Universal Robots PolyScope program: 05_var_local_01.urp

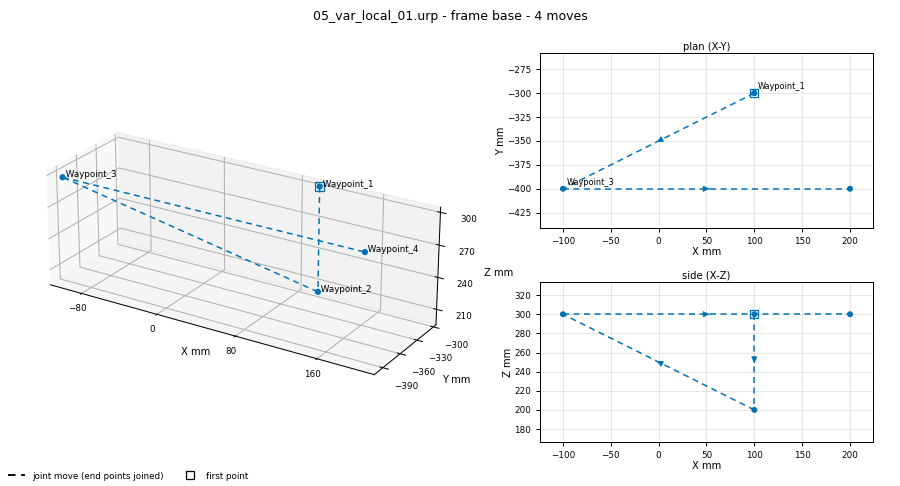
[picture p0: tool path of 05_var_local_01.urp in frame base, 4 of 4 moves have a stored position in this frame; points joined in program order, loops and branches not executed]
Program 05_var_local_01 (installation=default directory=/home/ur/ursim-current/programs/Test_Programs createdIn=5.9.1.1031110 lastSavedIn=5.9.1.1031110 robotSerialNumber=20195599999)
Calibrated DH parameters: a=[0, -0.425, -0.3922, 0, 0, 0]; d=[0.1625, 0, 0, 0.1333, 0.0997, 0.0996]; alpha=[1.570796, 0, 0, 1.570796, -1.570796, 0]; deltaTheta=[0, 0, 0, 0, 0, 0]
InitVariablesNode variables(variable(name=count, expression=0))
Robot Program (runOnlyOnce=false)
  MoveJ speed 60 deg/s, acceleration 80 deg/s^2 (useActiveTCP=true) feature=Base
    Waypoint Waypoint_1: TCP in base x=100 y=-300 z=300 mm, rx=0.0012 ry=3.1416 rz=0 rad; joints [-46.634, -65.64, -136.856, -67.504, 90, 43.412] deg
    Waypoint Waypoint_2: TCP in base x=100 y=-300 z=200 mm, rx=0 ry=3.1416 rz=0 rad; joints [-46.634, -77.892, -147.339, -44.768, 90, 43.366] deg
    count := count+1
    If count≟3
      MoveJ speed 60 deg/s, acceleration 80 deg/s^2 (useActiveTCP=true) feature=Base
        Waypoint Waypoint_3: TCP in base x=-100 y=-400 z=300 mm, rx=0 ry=3.1416 rz=0 rad; joints [-85.174, -82.459, -125.557, -61.984, 90, 4.826] deg
        Wait Sleep waitTime=1
    If count≟5
      MoveJ speed 60 deg/s, acceleration 80 deg/s^2 (useActiveTCP=true) feature=Base
        Waypoint Waypoint_4: TCP in base x=200 y=-400 z=300 mm, rx=0 ry=3.1416 rz=0 rad; joints [-46.093, -87.672, -120.896, -61.432, 90, 43.907] deg
        Popup Message (haltProgram=false message=Jop is done! inputType=Text)
        count := 0
